PROGRAM ST00_Sequence
VAR
END_VAR

END_PROGRAM

(* stored: Version 1.1.0.1, ProductVersion 3.1.4024.11
   POU ST00_Sequence: Id {025350f4-7dcb-4f6b-a07b-6c138f0e63d1}, SpecialFunc None *)
